// TIA Portal V20 export
// export: Created 2025-09-12T17:57:00.0000000Z, ExportSetting WithDefaults
TYPE "UDT300_EM_Heating"
   STRUCT
      High_Limit_DI : Bool;   // Digital Input: High-temperature limit switch (`True` = Fault).
      Heat_Stage1_Cmd_DO : Bool;   // Digital Output: Command for heating stage 1.
      High_Limit_Alm : Bool;   // Alarm: High-temperature limit fault.
   END_STRUCT;
END_TYPE
